FUNCTION_BLOCK alternative (* Basic Function Block Type *)
  (* Standard: 61499-2 *)
  (* Version 0.0, 24/05/2016, Chen-Wei, nxtControl GmbH, Template *)
  PACKAGE Main;
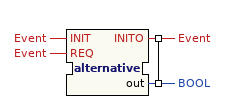
  EVENT_INPUT
    INIT; (* Initialization Request *)
    REQ;
  END_EVENT
  EVENT_OUTPUT
    INITO WITH out; (* Initialization Confirm *)
  END_EVENT
  VAR_OUTPUT
    out : BOOL; (* Output event qualifier *)
  END_VAR
  VAR
    internal : BOOL;
  END_VAR
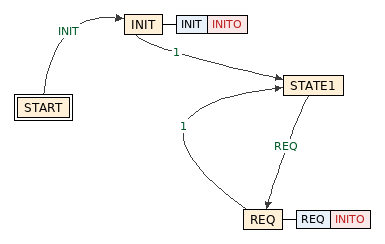
  EC_STATES
    START; (* Initial State *)
    INIT : INIT -> INITO; (* Initialization *)
    REQ : REQ -> INITO; (* Normal execution *)
    STATE1;
  END_STATES
  EC_TRANSITIONS
    START TO INIT := INIT;
    STATE1 TO REQ := REQ;
    REQ TO STATE1 := 1;
    INIT TO STATE1 := 1;
  END_TRANSITIONS
  ALGORITHM INIT IN ST: (* Initialization algorithm *)
out := TRUE;
internal := TRUE;

;
  END_ALGORITHM
  ALGORITHM REQ IN ST: (* Normally executed algorithm *)
REQ := 0;

internal := NOT internal;
out := internal;

;
  END_ALGORITHM
END_FUNCTION_BLOCK
